{attribute 'reflection'}
(* A small motor block with methods, an action and a property. *)
FUNCTION_BLOCK FB_Motor
VAR_INPUT
	enable : BOOL;
END_VAR
VAR_OUTPUT
	running : BOOL;
END_VAR
VAR
	speedSet : INT;
	startCount : DINT;
END_VAR

running := enable;
IF NOT running THEN
	speedSet := 0;
END_IF

METHOD PUBLIC Start : BOOL
VAR_INPUT
	force : BOOL;
END_VAR
startCount := startCount + 1;
Start := enable OR force;
END_METHOD

ACTION Reset:
running := FALSE;
startCount := 0;
END_ACTION

PROPERTY PUBLIC Speed : INT
GET
Speed := speedSet;
END_GET
SET
speedSet := Speed;
END_SET
END_PROPERTY

METHOD Stop
VAR
	wasRunning : BOOL;
END_VAR
wasRunning := running;
running := FALSE;
END_METHOD

END_FUNCTION_BLOCK

(* stored: Version 1.1.0.1, ProductVersion 3.1.4026.18
   POU FB_Motor: Id {00000000-0000-0000-0000-000000000030}, SpecialFunc None
   Method Start: Id {00000000-0000-0000-0000-000000000031}
   Action Reset: Id {00000000-0000-0000-0000-000000000032}
   Property Speed: Id {00000000-0000-0000-0000-000000000033}
   Get Get: Id {00000000-0000-0000-0000-000000000034}
   Set Set: Id {00000000-0000-0000-0000-000000000035}
   Method Stop: Id {00000000-0000-0000-0000-000000000036} *)
